// Mitsubishi GX Works2 project: 0630실린더 응용동작 4코멘트   PLC: Q02/Q02H

PROGRAM MAIN
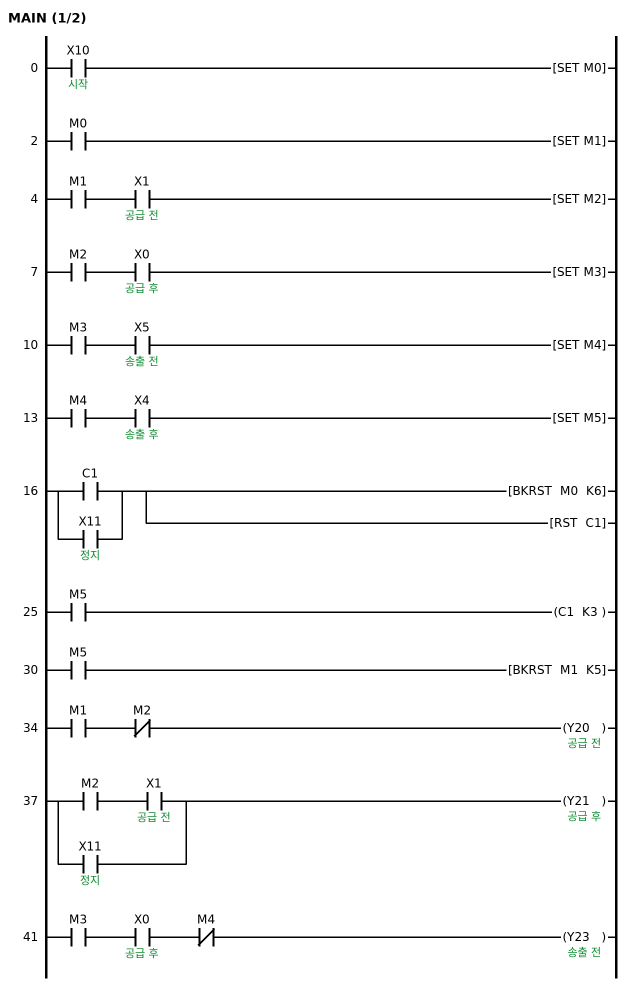
0     LD      X10  ; 시작
      SET     M0
2     LD      M0
      SET     M1
4     LD      M1
      AND     X1  ; 공급 전
      SET     M2
7     LD      M2
      AND     X0  ; 공급 후
      SET     M3
10    LD      M3
      AND     X5  ; 송출 전
      SET     M4
13    LD      M4
      AND     X4  ; 송출 후
      SET     M5
16    LD      C1
      OR      X11  ; 정지
      BKRST   M0 K6
      RST     C1
25    LD      M5
      OUT     C1 K3
30    LD      M5
      BKRST   M1 K5
34    LD      M1
      ANI     M2
      OUT     Y20  ; 공급 전
37    LD      M2
      AND     X1  ; 공급 전
      OR      X11  ; 정지
      OUT     Y21  ; 공급 후
41    LD      M3
      AND     X0  ; 공급 후
      ANI     M4
      OUT     Y23  ; 송출 전
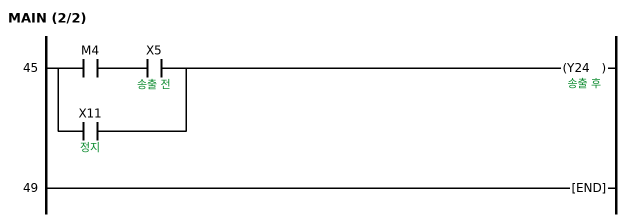
45    LD      M4
      AND     X5  ; 송출 전
      OR      X11  ; 정지
      OUT     Y24  ; 송출 후
49    END
END_PROGRAM

// device comments not shown above
X2  ; 드릴 상
X3  ; 드릴 하
X6  ; 배출 후
X7  ; 배출 전
Y22  ; 드릴 전
Y25  ; 배출 전
Y26  ; 배출 후
